Staubli VAL3: progItem.dtx

public InstrItem iEvent
  [0]
    string sType
    string sData
public string sID
